(* IEC 61131-3 sources: iec-checker/test/plcopen, 4 files *)

(* ---- cp1.st ---- *)
TYPE MyStruct:
STRUCT
    A : INT;
    B : INT;
END_STRUCT;
END_TYPE

FUNCTION FC_OffsetAccess : INT
VAR
    (* Map the STRUCTURE to a memory start address *)
    ms AT %MW500 : MyStruct;
    B_ByOffset: INT := 1;
END_VAR

(* Access B by offset(assume that %MW508 is the offset of B) *)
%MW508 := B_ByOffset;
(* Actually we should use ms.B like this: *)
(* ms.B := B_ByOffset; *)

END_FUNCTION

(* ---- cp3.st ---- *)
// 1 there is no init Violation
FUNCTION no_init_restart : INT
VAR
  some_var : INT;
END_VAR

(* Assuming some_var is 0 every time, which is dangerous *)
IF some_var > 5 THEN
  no_init_restart := some_var;
END_IF;

END_FUNCTION

// 2 there is no init Violation
FUNCTION Violation_DirectRead : INT
  VAR
    counter : INT := 0;
    some_var : INT; // Declared but not initialized
  END_VAR

  // Violation: some_var is read here for addition, but it has not been assigned
  counter := some_var + 1;

  some_var := 16#42;
  Violation_DirectRead := counter;
END_FUNCTION

// 3 there is no init Violation
FUNCTION Violation_Hidden : INT
  VAR
    counter : INT := 0;
    offset : INT;    // Forgot to initialize.
    base_val : INT := 100;
  END_VAR

  // Violation: although base_val has a value, offset is uninitialized
  counter := base_val + offset;

  Violation_Hidden := counter;
END_FUNCTION

// 4 all variables are initialized
FUNCTION Violation_None : INT
  VAR
    counter : INT := 0;
    offset : INT;    // Forgot to initialize.
    base_val : INT := 100;
  END_VAR

  offset := 42;
  counter := base_val + offset;

  Violation_None := counter;
END_FUNCTION

// 5 there is no init Violation
FUNCTION Violation_FuncCall1 : INT
  VAR
    counter : INT := 0;
    offset : INT;    // Forgot to initialize.
    base_val : INT := 100;
  END_VAR

  counter := func(base_val, offset);

  Violation_FuncCall1 := counter;
END_FUNCTION

// 6 there is no init Violation
FUNCTION Violation_FuncCall2 : INT
  VAR
    counter : INT := 0;
    offset : INT;    // Forgot to initialize.
    base_val : INT := 100;
  END_VAR
  (* In fact offset should not be alarmed here because offset is assigned but not used. *)
  counter := func(x:=base_val, y=>offset);

  Violation_FuncCall2 := counter;
END_FUNCTION

// 7 there is no Violation
FUNCTION Violation_FuncCall3 : INT
  VAR
    counter : INT := 0;
    offset : INT;
    base_val : INT := 100;
  END_VAR

  Violation_FuncCall3 := counter;
END_FUNCTION

// 8 there is Violation
FUNCTION Violation_FuncCall4 : INT
  VAR
    counter : INT := 0;
    offset : INT;
    base_val : INT := 100;
  END_VAR
  func(base_val, offset);
END_FUNCTION

// 9 there is Violation
FUNCTION Violation_self : INT
  VAR
    counter : INT := 0;
    offset : INT;
    base_val : INT := 100;
  END_VAR
  // offset := 1;
  offset := offset + 1;
END_FUNCTION

(* ---- cp8.st ---- *)
FUNCTION test1 : REAL
VAR
  a : REAL;
  b: REAL := 0.0;
END_VAR

IF b > 1.0 THEN
  a := 1.0;
END_IF;
test1 := a + b;
END_FUNCTION

// ---------------------------------------------

FUNCTION test2 : REAL
VAR
  a : REAL := 1.0;
  b: REAL := 1.0;
END_VAR

IF b = 0.0 THEN
  a := 1.0;
END_IF;
test2 := a + b;
END_FUNCTION

// ---------------------------------------------

FUNCTION test3 : REAL
VAR
  a : REAL := 1.0;
  b: REAL := 1.0;
END_VAR

IF b <> 0.0 THEN
  a := 1.0;
END_IF;
test3 := a + b;
END_FUNCTION

// ---------------------------------------------

FUNCTION test4 : REAL
VAR
  a : REAL := 1.0;
  b: REAL := 1.0;
END_VAR

IF b <> 1.0 THEN
  a := 1.0;
END_IF;
test4 := a + b;
END_FUNCTION

// ---------------------------------------------

FUNCTION test5 : REAL
VAR
  a : REAL := 1.0;
  b: REAL := 1.0;
END_VAR

IF b = 1.0 THEN
  a := 1.0;
END_IF;
test5 := a + b;
END_FUNCTION

// ---------------------------------------------

FUNCTION test6 : REAL
VAR
  a : REAL := 0.0;
  b: REAL := 1.0;
END_VAR

IF a = b THEN
  a := 1.0;
END_IF;
test6 := a + b;
END_FUNCTION

// ---------------------------------------------

FUNCTION test7 : REAL
VAR
  a : REAL := 0.0;
  b: REAL := 1.0;
END_VAR

IF a <> b THEN
  a := 1.0;
END_IF;
test7 := a + b;
END_FUNCTION

// ---------------------------------------------

FUNCTION test8 : REAL
VAR
  a : REAL := 1.0;
  b: REAL := 1.0;
END_VAR

IF a = b THEN
  a := 1.0;
ELSIF a <> b THEN
  a := 2.0;
END_IF;
test8 := a + b;

END_FUNCTION

// ---------------------------------------------

FUNCTION test9 : INT
VAR
  a : INT := 1;
  b: INT := 1;
END_VAR

IF INT_TO_REAL(a) <> INT_TO_REAL(b) THEN
  a := 2;
END_IF;
test9 := a + b;
END_FUNCTION

(* ---- cp2.st ---- *)
FUNCTION dead_code_after_return : INT
  VAR
    counter : INT := 0;
    some_var : INT;
  END_VAR
  counter := counter + 1;
  counter := 2 + 2;
  RETURN;
  some_var := SQRT(16#42); (* UnreachableCode error *)
  some_var := 16#42; (* No additional warnings *)
  some_var := 19;
END_FUNCTION

PROGRAM dead_code_in_the_loops
VAR a : INT; i : INT; END_VAR
  WHILE i < 10 DO
    IF i = 5 THEN
      i := i + 1;
      EXIT;
      i := 19; (* UnreachableCode error *)
      i := 42; (* No additional warnings *)
      i := 42;
    ELSIF i = 6 THEN
      CONTINUE;
      i := 3; (* UnreachableCode error *)
      i := 44; (* No additional warnings *)
      i := 19;
    END_IF;
    i := i + 2;
  END_WHILE;
  I := 0;
END_PROGRAM

FUNCTION FC_AlwaysTrue : INT
VAR_INPUT
    x : INT;
END_VAR

IF FALSE THEN
    FC_AlwaysTrue := x;
ELSE
    FC_AlwaysTrue := x + 100;   (* never executed *)
END_IF;

END_FUNCTION
